PROGRAM MAIN
VAR
END_VAR

GVL_ver.GCC2_xHV_DIS:=TRUE;
LadderLogic();
FB_KJL300();
FB_PBR260();
FB_TCP();

END_PROGRAM

(* stored: Version 1.1.0.1, ProductVersion 3.1.4022.3
   POU MAIN: Id {955730b6-e55e-459f-b0b3-a88c3048e89d}, SpecialFunc None *)
